FUNCTION_BLOCK LTimeOfDayPointerComparer EXTENDS Object IMPLEMENTS IPointerComparer
VAR
	_ClassName : STRING := __POUNAME();
END_VAR

{attribute 'monitoring' := 'call'}
PROPERTY ClassName : STRING
GET
ClassName := _ClassName;
END_GET
END_PROPERTY

{attribute "object_name" := "Compare"}
METHOD Compare : COMPARISION_RESULT
VAR_INPUT
	left : PVOID;
	right : PVOID;
END_VAR
VAR
	leftPointer : POINTER TO LTIME_OF_DAY; 
	rightPointer : POINTER TO LTIME_OF_DAY; 
END_VAR
IF left = 0 AND right = 0 THEN
	Compare := COMPARISION_RESULT.FIRST_EQUAL_TO_SECOND;
	RETURN;
END_IF

IF left = 0 THEN
	Compare := COMPARISION_RESULT.FIRST_LESS_THAN_SECOND;
	RETURN;	
END_IF

IF right = 0 THEN
	Compare := COMPARISION_RESULT.FIRST_GREATER_THAN_SECOND;
	RETURN;	
END_IF

leftPointer := left;
rightPointer := right;

IF leftPointer^ < rightPointer^ THEN
	Compare := COMPARISION_RESULT.FIRST_LESS_THAN_SECOND;
ELSIF leftPointer^ > rightPointer^ THEN
	Compare := COMPARISION_RESULT.FIRST_GREATER_THAN_SECOND;
ELSE
	Compare := COMPARISION_RESULT.FIRST_EQUAL_TO_SECOND;	
END_IF
END_METHOD

{attribute 'monitoring' := 'call'}
PROPERTY Size : ULINT
GET
Size := XSIZEOF(THIS^);
END_GET
END_PROPERTY

END_FUNCTION_BLOCK

(* stored: Version 1.1.0.1
   POU LTimeOfDayPointerComparer: Id {a86bbac2-4a38-4cd2-8777-a043f4d1467c}, SpecialFunc None
   Property ClassName: Id {70fc8c5d-3f6c-485a-9b2f-ff4a6b07319a}
   Get Get: Id {efa8db00-b2b6-4c11-a97c-704c4b295fc4}
   Method Compare: Id {906d60fa-f0d8-4f8d-9f44-c75d67ee6350}
   Property Size: Id {2f930264-531b-46d3-a470-bf71a7e8a0d5}
   Get Get: Id {4ca10f49-41a8-4758-80b5-ee7e152aa154} *)
